// TIA Portal V18 export
// export: Created 2025-12-01T12:38:50.4448398Z, ExportSetting None, DisplayName Totally Integrated Automation Portal, DisplayVersion V18 Update 5, DisplayName TIA Portal Openness, DisplayVersion V18 Update 5, DisplayName TIA Portal Teamcenter Gateway, DisplayVersion V18, DisplayName TIA Portal Version Control Interface, DisplayVersion V18, DisplayName STEP 7 Professional, DisplayVersion V18 Update 5, DisplayName STEP 7 Safety, DisplayVersion V18, DisplayName WinCC Professional, DisplayVersion V18 Update 5
DATA_BLOCK "Station_Sys"   // DB1060
TITLE = Station system DB
{ S7_Optimized_Access := 'FALSE' }
AUTHOR : RCS
FAMILY : Sys
VERSION : 2.0
// update 20160218
// stored: AutoNumber false
   VAR RETAIN
      ScreenNo : Int;   // For change HMI screen
      SpareB01 : Array[0..7] of Byte;   // *******************************************************************************
      Status : "RCS_SysStatus_V1";   // DBX10.0
      Input : Struct   // DBX20.0 For change PLC I input to PLC inside bit
         OP1 : Struct
            "Function 1" : Bool;
            "Function 2" : Bool;
            "Function 3" : Bool;
            "Function 4" : Bool;
            "Function 5" : Bool;
            "Function 6" : Bool;
            "Function 7" : Bool;
            "Function 8" : Bool;
         END_STRUCT;
         OP2 : Struct
            "Function 1" : Bool;
            "Function 2" : Bool;
            "Function 3" : Bool;
         END_STRUCT;
         OP3 : Struct
            "Function 1" : Bool;
            "Function 2" : Bool;
            "Function 3" : Bool;
         END_STRUCT;
      END_STRUCT;
      SpareB02 : Array[0..13] of Byte;   // *******************************************************************************
      HMI : Struct   // DBX40.0 HMI relation
         AP : Struct   // Area Pointer struct
            S1 : Int;
            CurrentScreenID : Int;
            S3 : Int;
            S4 : Int;
            S5 : Int;
         END_STRUCT;
      END_STRUCT;
      Cmd : "RCS_SysCmd_V1";   // DBX50.0
      SpareB03 : Array[0..7] of Byte;   // *******************************************************************************
      Interface : "RCS_SysComInterface_V1";   // DBX60.0
      SpareB04 : Array[0..3] of Byte;   // *******************************************************************************
      Initial : Struct   // DBX70.0
         Set : Bool;   // Trigger by HMI Button,[0]Total trigger
         Running : Bool;   // [0]Total initial Running
         OK : Bool;   // finish
      END_STRUCT;
      SpareB05 : Array[0..27] of Byte;   // *******************************************************************************
      Auto : "RCS_SysAuto_V1";   // DBX100.0
      SpareB10 : Array[0..5] of Byte;   // *******************************************************************************
      "A" : Struct   // DBX110.0 Auto control bit for some device
         "Device1 Auto control" : Bool;
         "Device2 Auto control" : Bool;
         "Device3 Auto control" : Bool;
         "Device4 Auto control" : Bool;
         "Device 01" : Struct
            "Function 1" : Bool;   // Flash
            "Function 2" : Bool;
            "Function 3" : Bool;   // Flash
         END_STRUCT;
         "Device 02" : Struct
            "Function 1" : Bool;   // Flash
            "Function 2" : Bool;
            "Function 3" : Bool;   // Flash
         END_STRUCT;
      END_STRUCT;
      SpareB11 : Array[0..33] of Byte;   // *******************************************************************************
      Manual : "RCS_SysManual_V1";   // DBX150.0
      SpareB12 : Array[0..6] of Byte;   // *******************************************************************************
      "M" : Struct   // DBX160.0 Manual control bit for some device
         "Device1 Manual control" : Bool;
         "Device2 Manual control" : Bool;
         "Device3 Manual control" : Bool;
         "Device4 Manual control" : Bool;
      END_STRUCT;
      SpareB13 : Array[0..37] of Byte;   // *******************************************************************************
      Safety : "RCS_SysSafety_V1";   // DBX200.0
      SpareB20 : Array[0..9] of Byte;   // *******************************************************************************
      Signal : Struct   // DBX220.0
         MainPressureSwitch1 : Bool;
         MainPressureSwitch2 : Bool;
         MainPressureSwitch3 : Bool;
      END_STRUCT;
      SpareB21 : Array[0..36] of Byte;   // *******************************************************************************
      Flag : Struct   // DBX260.0
         Processstart : Bool;
         PeocessComplete : Bool;
         IndexTable : Struct
            Interlock : Bool;
            TableRunning : Bool;   // Complete cycle Running
            StopandPosition : Bool;
            PositionOK : Bool;
            PositionNG : Bool;
            FixtureOK : Bool;
            FixtureNG : Bool;
            InitialOK : Bool;
         END_STRUCT;
      END_STRUCT;
      SpareB22 : Array[0..5] of Byte;   // *******************************************************************************
      P : Struct   // Positive RLO Edge Detection:-(P)- DBX270
         Record : Bool;
         "Set index run" : Bool;
         initial : Array[0..7] of Bool;
      END_STRUCT;
      SpareB23 : Array[0..5] of Byte;   // *******************************************************************************
      N : Struct   // Negative RLO Edge Detection:-(N)- DBX280
         Spare : Bool;
      END_STRUCT;
      SpareB24 : Array[0..17] of Byte;   // *******************************************************************************
      Alarm : "RCS_SysAlarmWarning_V1";   // DBX300.0
      SpareB30 : Array[0..7] of Byte;   // *******************************************************************************
      Warning : "RCS_SysAlarmWarning_V1";   // DBX310.0 / DBX500.0
      SpareB31 : Array[0..7] of Byte;   // *******************************************************************************
      AlarmTimes : Struct   // DBX320 If a fault continue happened over Limit times, than Auto running will be stopped / If a fault continue happened over Limit_times，Auto running will be stopped
         ForceStop : Bool;   // DBX320.0 / DBX650.0
         Reset : Bool;
         Limit : Int;
      END_STRUCT;
      SpareB33 : Array[0..5] of Byte;   // *******************************************************************************
      AlarmWarning : Int;   // DBX330 1:Alarm 2:Warning / DBX660 1:Alarm 2:Warning
      SpareB34 : Array[0..17] of Byte;   // *******************************************************************************
      Count : "RCS_SysCount_V1";   // DBX350.0 / DBX700.0
      SpareB40 : Array[0..11] of Byte;   // *******************************************************************************
      TotalCycleTime : "RCS_SysCycleTime_V1";   // DBX500.0 / DBX850.0
      SpareB41 : Array[0..11] of Byte;   // *******************************************************************************
      MachineCycleTime : "RCS_SysCycleTime_V1";   // DBX600.0 / DBX950.0
      SpareB42 : Array[0..11] of Byte;   // *******************************************************************************
      UserName { S7_SetPoint := 'True'} : String[20];   // DBX700.0
   END_VAR
BEGIN
   // Cmd.Record : 记录
   // Cmd.BuzzerOn : 蜂鸣器 On
   Cmd.OnOffLine := TRUE;
END_DATA_BLOCK
